// TIA Portal project "Xulynuocthai" (V16)

(* hardware
DEVICE "S7-1200 station_1"  S7-1200 Station
   slot 0: "Rack_0"  S7-1200 Rack  Rack  V1.0
   slot 1: "PLC_1"  CPU 1212C DC/DC/DC  6ES7 212-1AE40-0XB0  V4.4
*)

// ===== PLC "PLC_1"  CPU 1212C DC/DC/DC =====

VAR_GLOBAL   // PLC tag table "Default tag table"
   "M_Xung" AT %M20.0 : Bool;
   "M_ClosePump12" AT %M30.0 : Bool;
   "M_Close_Pump3" AT %M30.1 : Bool;
   "M_Close_Valves1" AT %M30.2 : Bool;
   "M_Close_Valver2" AT %M30.3 : Bool;
   "M_Remember" AT %MW100 : Int;
   "M_Enable_CloseP12" AT %M30.4 : Bool;
   "M_Enable_CloseP3" AT %M30.5 : Bool;
   "M_Enable_CloseV1" AT %M31.2 : Bool;
   "M_Enable_CloseV2" AT %M31.3 : Bool;
END_VAR

DATA_BLOCK "ReceiveData"   // DB2
{ S7_Optimized_Access := 'FALSE' }
VERSION : 0.1
   VAR
      I_SystemOn : Bool;
      I_SystemOff : Bool;
      I_Tank1_ssLow : Bool;
      I_Tank1_ssHigh : Bool;
      I_Tank2_ssLow : Bool;
      I_Tank2_ssHigh : Bool;
      I_Tank3_ssLow : Bool;
      I_Tank3_sHigh : Bool;
      I_Tank4_ssLow : Bool;
      I_Tank4_ssHigh : Bool;
      Q_Pump1 : Bool;
      Q_Pump2 : Bool;
      Q_Pump3 : Bool;
      Q_Pump4 : Bool;
      Q_Valves1 : Bool;
      Q_Valves2 : Bool;
      Q_Lamp_System : Bool;
      Set_Salt_Value : Real;
      Set_Time_Luanphien : Int;
      Act_Salt_Value : Real;
      Act_Time_Min : Int;
      Act_Time_Sec : Int;
      Set_Xung : DInt;
   END_VAR
BEGIN
END_DATA_BLOCK

// folder: System blocks/Program resources

DATA_BLOCK "Xung"   // DB1
{ S7_Optimized_Access := 'TRUE' }
AUTHOR : Simatic
FAMILY : IEC
NAME : IEC_TMR
VERSION : 1.0
// stored: InstanceOfName IEC_TIMER
"IEC_TIMER"
BEGIN
END_DATA_BLOCK

// folder: (top level)

ORGANIZATION_BLOCK "Main"   // OB1, LAD, ProgramCycle
TITLE = "Main Program Sweep (Cycle)"
{ S7_Optimized_Access := 'TRUE' }
VERSION : 0.1
   VAR_INPUT
      Initial_Call : Bool;   // Initial call of this OB
      Remanence : Bool;   // =True, if remanent data are available
   END_VAR
   VAR_TEMP   // added for the SCL form of the ladder/FBD networks
      _w1 : Bool;
      _w2 : Bool;
   END_VAR
BEGIN

REGION Network 1
   // on/off hệ thống
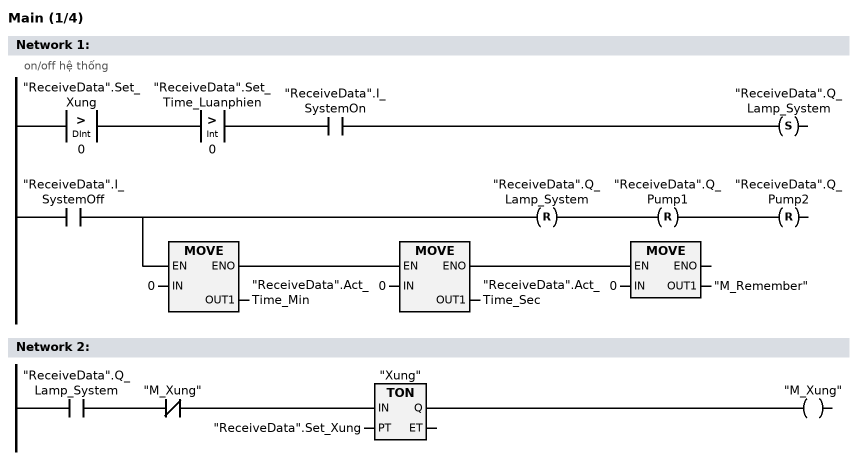
   RUNG wire#powerrail
      { S7_Templates := "SrcType := DInt" } GT_Contact(in1 := "ReceiveData".Set_Xung, in2 := 0)
      { S7_Templates := "SrcType := Int" } GT_Contact(in1 := "ReceiveData".Set_Time_Luanphien, in2 := 0)
      Contact( "ReceiveData".I_SystemOn )
      S_Coil( "ReceiveData".Q_Lamp_System )
   END_RUNG
   RUNG wire#powerrail
      Contact( "ReceiveData".I_SystemOff )
      wire#w1
      R_Coil( "ReceiveData".Q_Lamp_System )
      R_Coil( "ReceiveData".Q_Pump1 )
      R_Coil( "ReceiveData".Q_Pump2 )
   END_RUNG
   RUNG wire#w1
      Move(in := 0, out1 => "ReceiveData".Act_Time_Min)
      Move(in := 0, out1 => "ReceiveData".Act_Time_Sec)
      Move(in := 0, out1 => "M_Remember")
   END_RUNG
   // the same network as SCL:
   IF ("ReceiveData".Set_Xung > 0) AND ("ReceiveData".Set_Time_Luanphien > 0) AND "ReceiveData".I_SystemOn THEN
       "ReceiveData".Q_Lamp_System := TRUE;
   END_IF;
   IF "ReceiveData".I_SystemOff THEN
       "ReceiveData".Q_Lamp_System := FALSE;
       "ReceiveData".Q_Pump1 := FALSE;
       "ReceiveData".Q_Pump2 := FALSE;
       "ReceiveData".Act_Time_Min := 0;
       "ReceiveData".Act_Time_Sec := 0;
       "M_Remember" := 0;
   END_IF;
END_REGION

REGION Network 2
   "Xung".TON(IN := "ReceiveData".Q_Lamp_System AND NOT "M_Xung", PT := "ReceiveData".Set_Xung);
   "M_Xung" := "Xung".Q;
END_REGION

REGION Network 3: Bowm1,2 luân phiên hoạt động
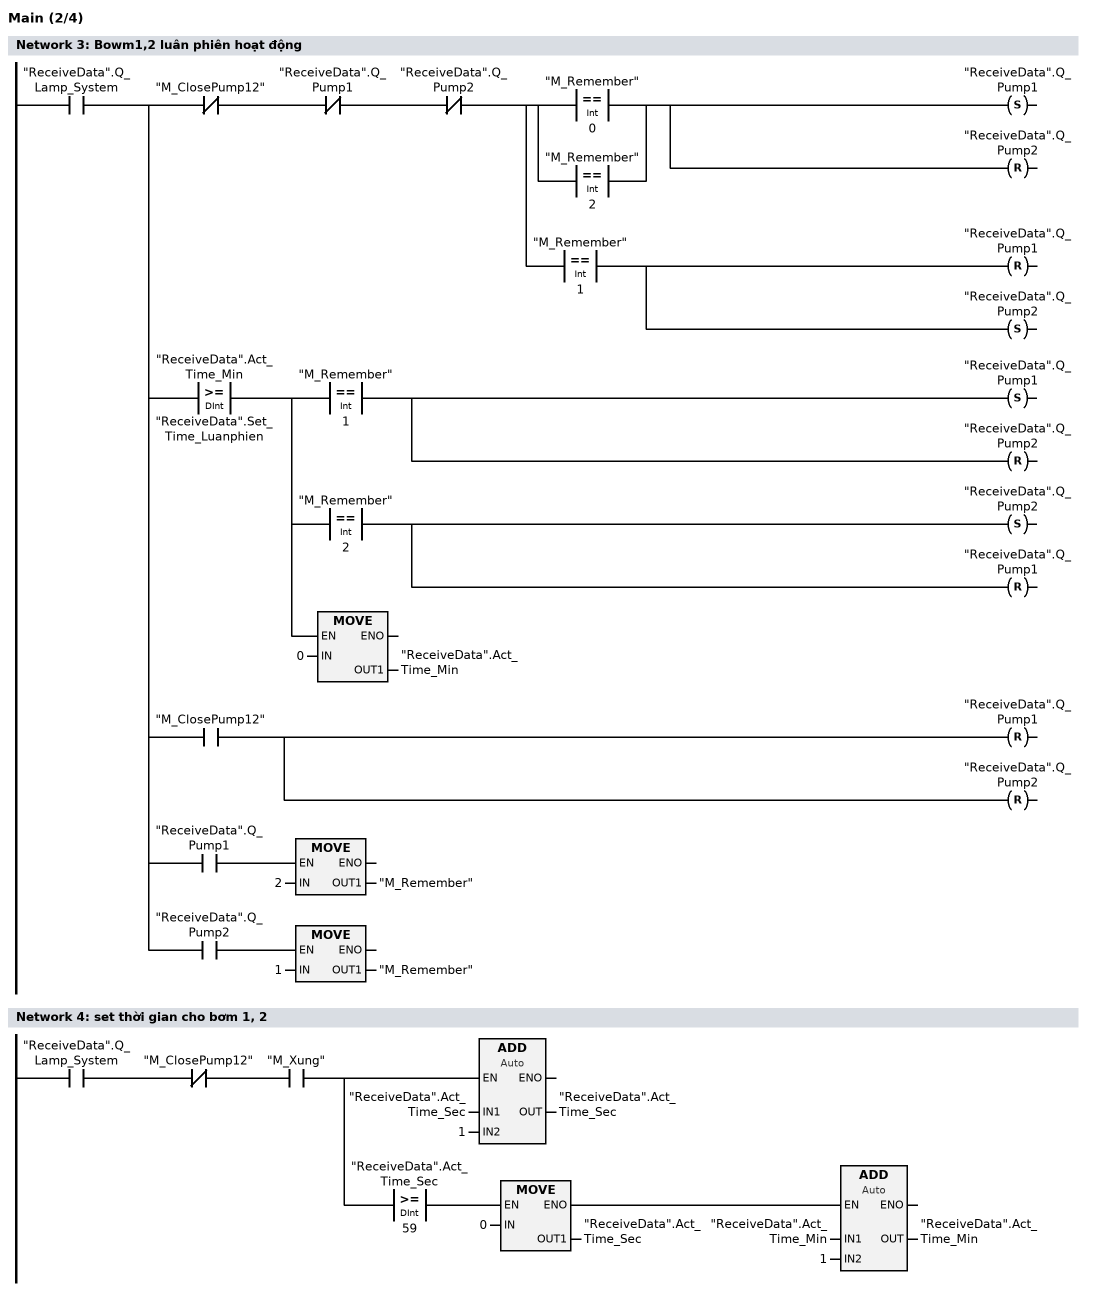
   RUNG wire#powerrail
      Contact( "ReceiveData".Q_Lamp_System )
      wire#w1
      I_Contact( "M_ClosePump12" )
      I_Contact( "ReceiveData".Q_Pump1 )
      I_Contact( "ReceiveData".Q_Pump2 )
      wire#w2
      { S7_Templates := "SrcType := Int" } EQ_Contact(in1 := "M_Remember", in2 := 0)
      wire#w3
      S_Coil( "ReceiveData".Q_Pump1 )
   END_RUNG
   RUNG wire#w2
      { S7_Templates := "SrcType := Int" } EQ_Contact(in1 := "M_Remember", in2 := 2)
   END_RUNG wire#w3
   RUNG wire#w3
      R_Coil( "ReceiveData".Q_Pump2 )
   END_RUNG
   RUNG wire#w2
      { S7_Templates := "SrcType := Int" } EQ_Contact(in1 := "M_Remember", in2 := 1)
      wire#w4
      R_Coil( "ReceiveData".Q_Pump1 )
   END_RUNG
   RUNG wire#w4
      S_Coil( "ReceiveData".Q_Pump2 )
   END_RUNG
   RUNG wire#w1
      { S7_Templates := "SrcType := DInt" } GE_Contact(in1 := "ReceiveData".Act_Time_Min, in2 := "ReceiveData".Set_Time_Luanphien)
      wire#w5
      { S7_Templates := "SrcType := Int" } EQ_Contact(in1 := "M_Remember", in2 := 1)
      wire#w6
      S_Coil( "ReceiveData".Q_Pump1 )
   END_RUNG
   RUNG wire#w6
      R_Coil( "ReceiveData".Q_Pump2 )
   END_RUNG
   RUNG wire#w5
      { S7_Templates := "SrcType := Int" } EQ_Contact(in1 := "M_Remember", in2 := 2)
      wire#w7
      S_Coil( "ReceiveData".Q_Pump2 )
   END_RUNG
   RUNG wire#w7
      R_Coil( "ReceiveData".Q_Pump1 )
   END_RUNG
   RUNG wire#w5
      Move(in := 0, out1 => "ReceiveData".Act_Time_Min)
   END_RUNG
   RUNG wire#w1
      Contact( "M_ClosePump12" )
      wire#w8
      R_Coil( "ReceiveData".Q_Pump1 )
   END_RUNG
   RUNG wire#w8
      R_Coil( "ReceiveData".Q_Pump2 )
   END_RUNG
   RUNG wire#w1
      Contact( "ReceiveData".Q_Pump1 )
      Move(in := 2, out1 => "M_Remember")
   END_RUNG
   RUNG wire#w1
      Contact( "ReceiveData".Q_Pump2 )
      Move(in := 1, out1 => "M_Remember")
   END_RUNG
   // the same network as SCL:
   #_w1 := "ReceiveData".Q_Lamp_System AND NOT "M_ClosePump12" AND NOT "ReceiveData".Q_Pump1 AND NOT "ReceiveData".Q_Pump2;
   IF #_w1 AND (("M_Remember" = 0) OR ("M_Remember" = 2)) THEN
       "ReceiveData".Q_Pump1 := TRUE;
       "ReceiveData".Q_Pump2 := FALSE;
   END_IF;
   IF #_w1 AND ("M_Remember" = 1) THEN
       "ReceiveData".Q_Pump1 := FALSE;
       "ReceiveData".Q_Pump2 := TRUE;
   END_IF;
   #_w2 := "ReceiveData".Q_Lamp_System AND ("ReceiveData".Act_Time_Min >= "ReceiveData".Set_Time_Luanphien);
   IF #_w2 AND ("M_Remember" = 1) THEN
       "ReceiveData".Q_Pump1 := TRUE;
       "ReceiveData".Q_Pump2 := FALSE;
   END_IF;
   IF #_w2 AND ("M_Remember" = 2) THEN
       "ReceiveData".Q_Pump2 := TRUE;
       "ReceiveData".Q_Pump1 := FALSE;
   END_IF;
   IF #_w2 THEN "ReceiveData".Act_Time_Min := 0; END_IF;
   IF "ReceiveData".Q_Lamp_System AND "M_ClosePump12" THEN
       "ReceiveData".Q_Pump1 := FALSE;
       "ReceiveData".Q_Pump2 := FALSE;
   END_IF;
   IF "ReceiveData".Q_Lamp_System AND "ReceiveData".Q_Pump1 THEN "M_Remember" := 2; END_IF;
   IF "ReceiveData".Q_Lamp_System AND "ReceiveData".Q_Pump2 THEN "M_Remember" := 1; END_IF;
END_REGION

REGION Network 4: set thời gian cho bơm 1, 2
   RUNG wire#powerrail
      Contact( "ReceiveData".Q_Lamp_System )
      I_Contact( "M_ClosePump12" )
      Contact( "M_Xung" )
      wire#w1
      Add(in1 := "ReceiveData".Act_Time_Sec, in2 := 1, out => "ReceiveData".Act_Time_Sec)
   END_RUNG
   RUNG wire#w1
      { S7_Templates := "SrcType := DInt" } GE_Contact(in1 := "ReceiveData".Act_Time_Sec, in2 := 59)
      Move(in := 0, out1 => "ReceiveData".Act_Time_Sec)
      Add(in1 := "ReceiveData".Act_Time_Min, in2 := 1, out => "ReceiveData".Act_Time_Min)
   END_RUNG
   // the same network as SCL:
   #_w1 := "ReceiveData".Q_Lamp_System AND NOT "M_ClosePump12" AND "M_Xung";
   IF #_w1 THEN "ReceiveData".Act_Time_Sec := "ReceiveData".Act_Time_Sec + 1; END_IF;
   #_w2 := #_w1 AND ("ReceiveData".Act_Time_Sec >= 59);
   IF #_w2 THEN
       "ReceiveData".Act_Time_Sec := 0;
       "ReceiveData".Act_Time_Min := "ReceiveData".Act_Time_Min + 1;
   END_IF;
END_REGION

REGION Network 5: đóng bơm 1,2
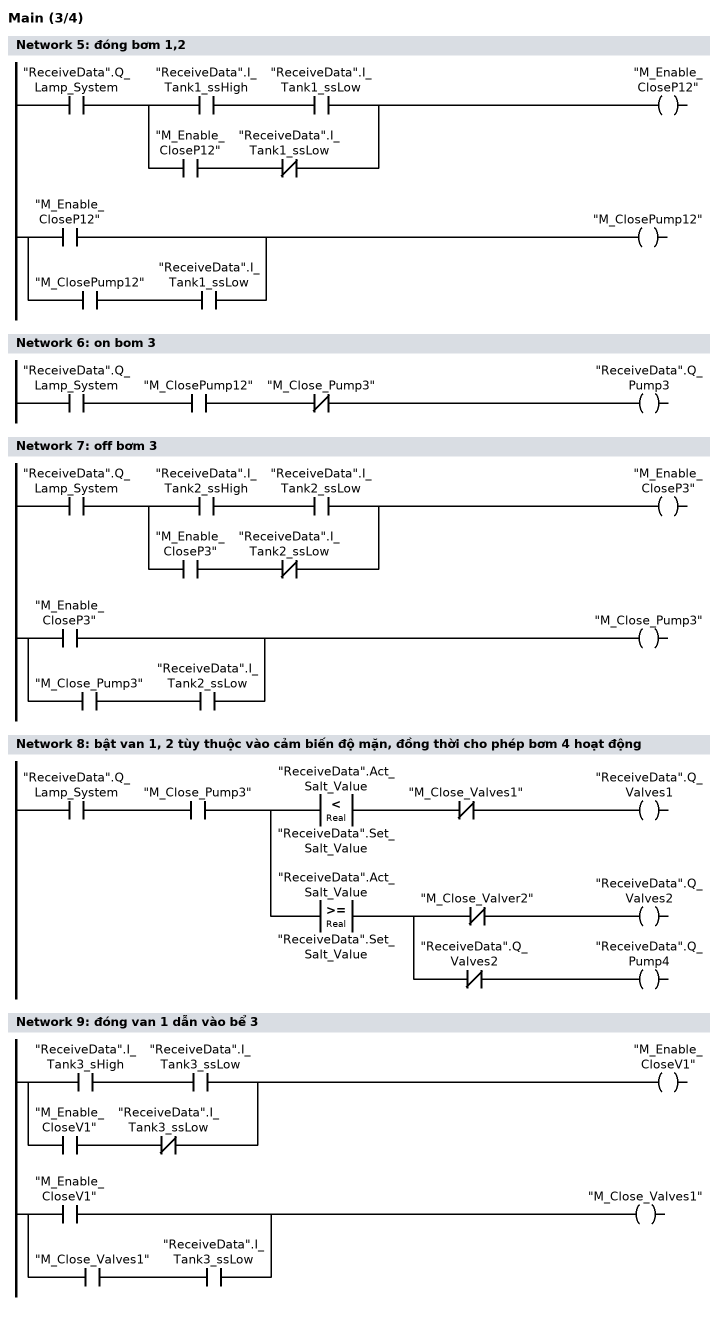
   RUNG wire#powerrail
      Contact( "ReceiveData".Q_Lamp_System )
      wire#w1
      Contact( "ReceiveData".I_Tank1_ssHigh )
      Contact( "ReceiveData".I_Tank1_ssLow )
      wire#w2
      Coil( "M_Enable_CloseP12" )
   END_RUNG
   RUNG wire#w1
      Contact( "M_Enable_CloseP12" )
      I_Contact( "ReceiveData".I_Tank1_ssLow )
   END_RUNG wire#w2
   RUNG wire#powerrail
      Contact( "M_Enable_CloseP12" )
      wire#w3
      Coil( "M_ClosePump12" )
   END_RUNG
   RUNG wire#powerrail
      Contact( "M_ClosePump12" )
      Contact( "ReceiveData".I_Tank1_ssLow )
   END_RUNG wire#w3
   // the same network as SCL:
   "M_Enable_CloseP12" := "ReceiveData".Q_Lamp_System AND (("ReceiveData".I_Tank1_ssHigh AND "ReceiveData".I_Tank1_ssLow) OR ("M_Enable_CloseP12" AND NOT "ReceiveData".I_Tank1_ssLow));
   "M_ClosePump12" := "M_Enable_CloseP12" OR ("M_ClosePump12" AND "ReceiveData".I_Tank1_ssLow);
END_REGION

REGION Network 6: on bom 3
   RUNG wire#powerrail
      Contact( "ReceiveData".Q_Lamp_System )
      Contact( "M_ClosePump12" )
      I_Contact( "M_Close_Pump3" )
      Coil( "ReceiveData".Q_Pump3 )
   END_RUNG
   // the same network as SCL:
   "ReceiveData".Q_Pump3 := "ReceiveData".Q_Lamp_System AND "M_ClosePump12" AND NOT "M_Close_Pump3";
END_REGION

REGION Network 7: off bơm 3
   RUNG wire#powerrail
      Contact( "ReceiveData".Q_Lamp_System )
      wire#w1
      Contact( "ReceiveData".I_Tank2_ssHigh )
      Contact( "ReceiveData".I_Tank2_ssLow )
      wire#w2
      Coil( "M_Enable_CloseP3" )
   END_RUNG
   RUNG wire#w1
      Contact( "M_Enable_CloseP3" )
      I_Contact( "ReceiveData".I_Tank2_ssLow )
   END_RUNG wire#w2
   RUNG wire#powerrail
      Contact( "M_Enable_CloseP3" )
      wire#w3
      Coil( "M_Close_Pump3" )
   END_RUNG
   RUNG wire#powerrail
      Contact( "M_Close_Pump3" )
      Contact( "ReceiveData".I_Tank2_ssLow )
   END_RUNG wire#w3
   // the same network as SCL:
   "M_Enable_CloseP3" := "ReceiveData".Q_Lamp_System AND (("ReceiveData".I_Tank2_ssHigh AND "ReceiveData".I_Tank2_ssLow) OR ("M_Enable_CloseP3" AND NOT "ReceiveData".I_Tank2_ssLow));
   "M_Close_Pump3" := "M_Enable_CloseP3" OR ("M_Close_Pump3" AND "ReceiveData".I_Tank2_ssLow);
END_REGION

REGION Network 8: bật van 1, 2 tùy thuộc vào cảm biến độ mặn, đồng thời cho phép bơm 4 hoạt động
   RUNG wire#powerrail
      Contact( "ReceiveData".Q_Lamp_System )
      Contact( "M_Close_Pump3" )
      wire#w1
      { S7_Templates := "SrcType := Real" } LT_Contact(in1 := "ReceiveData".Act_Salt_Value, in2 := "ReceiveData".Set_Salt_Value)
      I_Contact( "M_Close_Valves1" )
      Coil( "ReceiveData".Q_Valves1 )
   END_RUNG
   RUNG wire#w1
      { S7_Templates := "SrcType := Real" } GE_Contact(in1 := "ReceiveData".Act_Salt_Value, in2 := "ReceiveData".Set_Salt_Value)
      wire#w2
      I_Contact( "M_Close_Valver2" )
      Coil( "ReceiveData".Q_Valves2 )
   END_RUNG
   RUNG wire#w2
      I_Contact( "ReceiveData".Q_Valves2 )
      Coil( "ReceiveData".Q_Pump4 )
   END_RUNG
   // the same network as SCL:
   #_w1 := "ReceiveData".Q_Lamp_System AND "M_Close_Pump3";
   "ReceiveData".Q_Valves1 := #_w1 AND ("ReceiveData".Act_Salt_Value < "ReceiveData".Set_Salt_Value) AND NOT "M_Close_Valves1";
   #_w2 := #_w1 AND ("ReceiveData".Act_Salt_Value >= "ReceiveData".Set_Salt_Value);
   "ReceiveData".Q_Valves2 := #_w2 AND NOT "M_Close_Valver2";
   "ReceiveData".Q_Pump4 := #_w2 AND NOT "ReceiveData".Q_Valves2;
END_REGION

REGION Network 9: đóng van 1 dẫn vào bể 3
   RUNG wire#powerrail
      Contact( "ReceiveData".I_Tank3_sHigh )
      Contact( "ReceiveData".I_Tank3_ssLow )
      wire#w1
      Coil( "M_Enable_CloseV1" )
   END_RUNG
   RUNG wire#powerrail
      Contact( "M_Enable_CloseV1" )
      I_Contact( "ReceiveData".I_Tank3_ssLow )
   END_RUNG wire#w1
   RUNG wire#powerrail
      Contact( "M_Enable_CloseV1" )
      wire#w2
      Coil( "M_Close_Valves1" )
   END_RUNG
   RUNG wire#powerrail
      Contact( "M_Close_Valves1" )
      Contact( "ReceiveData".I_Tank3_ssLow )
   END_RUNG wire#w2
   // the same network as SCL:
   "M_Enable_CloseV1" := ("ReceiveData".I_Tank3_sHigh AND "ReceiveData".I_Tank3_ssLow) OR ("M_Enable_CloseV1" AND NOT "ReceiveData".I_Tank3_ssLow);
   "M_Close_Valves1" := "M_Enable_CloseV1" OR ("M_Close_Valves1" AND "ReceiveData".I_Tank3_ssLow);
END_REGION

REGION Network 10: đóng van 2 dẫn vào bể 4
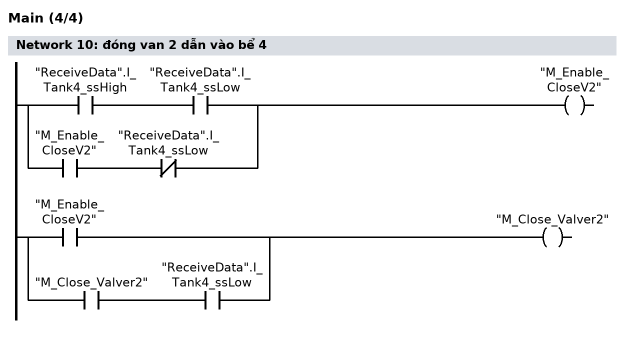
   RUNG wire#powerrail
      Contact( "ReceiveData".I_Tank4_ssHigh )
      Contact( "ReceiveData".I_Tank4_ssLow )
      wire#w1
      Coil( "M_Enable_CloseV2" )
   END_RUNG
   RUNG wire#powerrail
      Contact( "M_Enable_CloseV2" )
      I_Contact( "ReceiveData".I_Tank4_ssLow )
   END_RUNG wire#w1
   RUNG wire#powerrail
      Contact( "M_Enable_CloseV2" )
      wire#w2
      Coil( "M_Close_Valver2" )
   END_RUNG
   RUNG wire#powerrail
      Contact( "M_Close_Valver2" )
      Contact( "ReceiveData".I_Tank4_ssLow )
   END_RUNG wire#w2
   // the same network as SCL:
   "M_Enable_CloseV2" := ("ReceiveData".I_Tank4_ssHigh AND "ReceiveData".I_Tank4_ssLow) OR ("M_Enable_CloseV2" AND NOT "ReceiveData".I_Tank4_ssLow);
   "M_Close_Valver2" := "M_Enable_CloseV2" OR ("M_Close_Valver2" AND "ReceiveData".I_Tank4_ssLow);
END_REGION
END_ORGANIZATION_BLOCK